// TIA Portal project "btvn_tuan2_light_traffic_2_chieu" (V14)

(* hardware
DEVICE "S7-1200 station_1"  S7-1200 Station
   slot 0: "Rack_0"  S7-1200 Rack  Rack  V1.0
   slot 1: "PLC_1"  CPU 1214C DC/DC/DC  6ES7 214-1AG40-0XB0  V4.2
DEVICE "HMI_1"  KTP700 Basic PN
   slot 0: "KTP700 Basic PN"  KTP700 Basic PN  6AV2 123-2GB03-0AX0  14.0.1.0
   slot 1: "HMI_RT_1"  KTP700 Basic PN  6AV2 123-2GB03-0AX0  14.0.1.0
   slot 5: "HMI_1.IE_CP_1"  PROFINET Interface  14.0.1.0
      slot 1: "PROFINET Interface_1"  PROFINET Interface
         slot 1: "Port_1"  Port
*)

// ===== PLC "PLC_1"  CPU 1214C DC/DC/DC =====

VAR_GLOBAL   // PLC tag table "Default tag table"
   "start" AT %M0.0 : Bool;
   "return" AT %M0.1 : Bool;
   "A do1" AT %M1.0 : Bool;
   "A vang1" AT %M1.2 : Bool;
   "A xanh 1" AT %M1.3 : Bool;
   "B do" AT %M0.5 : Bool;
   "B vang" AT %M0.6 : Bool;
   "B xanh" AT %M0.7 : Bool;
   "sleep mode" AT %I0.2 : Bool;
   "uu tien mode" AT %M1.1 : Bool;
   "uu tien 1" AT %I0.0 : Bool;
   "uu tien 2" AT %I0.1 : Bool;
   "tmp" AT %M1.4 : Bool;
   "tmp(1)" AT %M1.5 : Bool;
   "save2" AT %M1.6 : Bool;
   "save1" AT %M1.7 : Bool;
   "A vang 2" AT %M0.2 : Bool;
   "A xanh 2" AT %M0.3 : Bool;
   "A do 2" AT %M0.4 : Bool;
   "Tag_1" AT %Q0.2 : Bool;
   "Tag_2" AT %Q0.0 : Bool;
   "Tag_3" AT %Q0.1 : Bool;
   "Tag_4" AT %Q0.3 : Bool;
END_VAR

// folder: System blocks/Program resources

DATA_BLOCK "IEC_Timer_0_DB"   // DB1
{ S7_Optimized_Access := 'TRUE' }
AUTHOR : Simatic
FAMILY : IEC
NAME : IEC_TMR
VERSION : 1.0
// stored: InstanceOfName IEC_TIMER
"IEC_TIMER"
BEGIN
END_DATA_BLOCK

DATA_BLOCK "IEC_Timer_0_DB_1"   // DB2
{ S7_Optimized_Access := 'TRUE' }
AUTHOR : Simatic
FAMILY : IEC
NAME : IEC_TMR
VERSION : 1.0
// stored: InstanceOfName IEC_TIMER
"IEC_TIMER"
BEGIN
END_DATA_BLOCK

DATA_BLOCK "IEC_Timer_0_DB_2"   // DB3
{ S7_Optimized_Access := 'TRUE' }
AUTHOR : Simatic
FAMILY : IEC
NAME : IEC_TMR
VERSION : 1.0
// stored: InstanceOfName IEC_TIMER
"IEC_TIMER"
BEGIN
END_DATA_BLOCK

DATA_BLOCK "IEC_Timer_0_DB_3"   // DB4
{ S7_Optimized_Access := 'TRUE' }
AUTHOR : Simatic
FAMILY : IEC
NAME : IEC_TMR
VERSION : 1.0
// stored: InstanceOfName IEC_TIMER
"IEC_TIMER"
BEGIN
END_DATA_BLOCK

DATA_BLOCK "IEC_Timer_0_DB_4"   // DB5
{ S7_Optimized_Access := 'TRUE' }
AUTHOR : Simatic
FAMILY : IEC
NAME : IEC_TMR
VERSION : 1.0
// stored: InstanceOfName IEC_TIMER
"IEC_TIMER"
BEGIN
END_DATA_BLOCK

DATA_BLOCK "IEC_Timer_0_DB_5"   // DB6
{ S7_Optimized_Access := 'TRUE' }
AUTHOR : Simatic
FAMILY : IEC
NAME : IEC_TMR
VERSION : 1.0
// stored: InstanceOfName IEC_TIMER
"IEC_TIMER"
BEGIN
END_DATA_BLOCK

// folder: (top level)

ORGANIZATION_BLOCK "Main"   // OB1, LAD, ProgramCycle
TITLE = "Main Program Sweep (Cycle)"
{ S7_Optimized_Access := 'TRUE' }
VERSION : 0.1
   VAR_INPUT
      Initial_Call : Bool;   // Initial call of this OB
      Remanence : Bool;   // =True, if remanent data are available
   END_VAR
   VAR_TEMP   // added for the SCL form of the ladder/FBD networks
      _w1 : Bool;
   END_VAR
BEGIN

REGION Network 1: tuan tu sinh ra state den
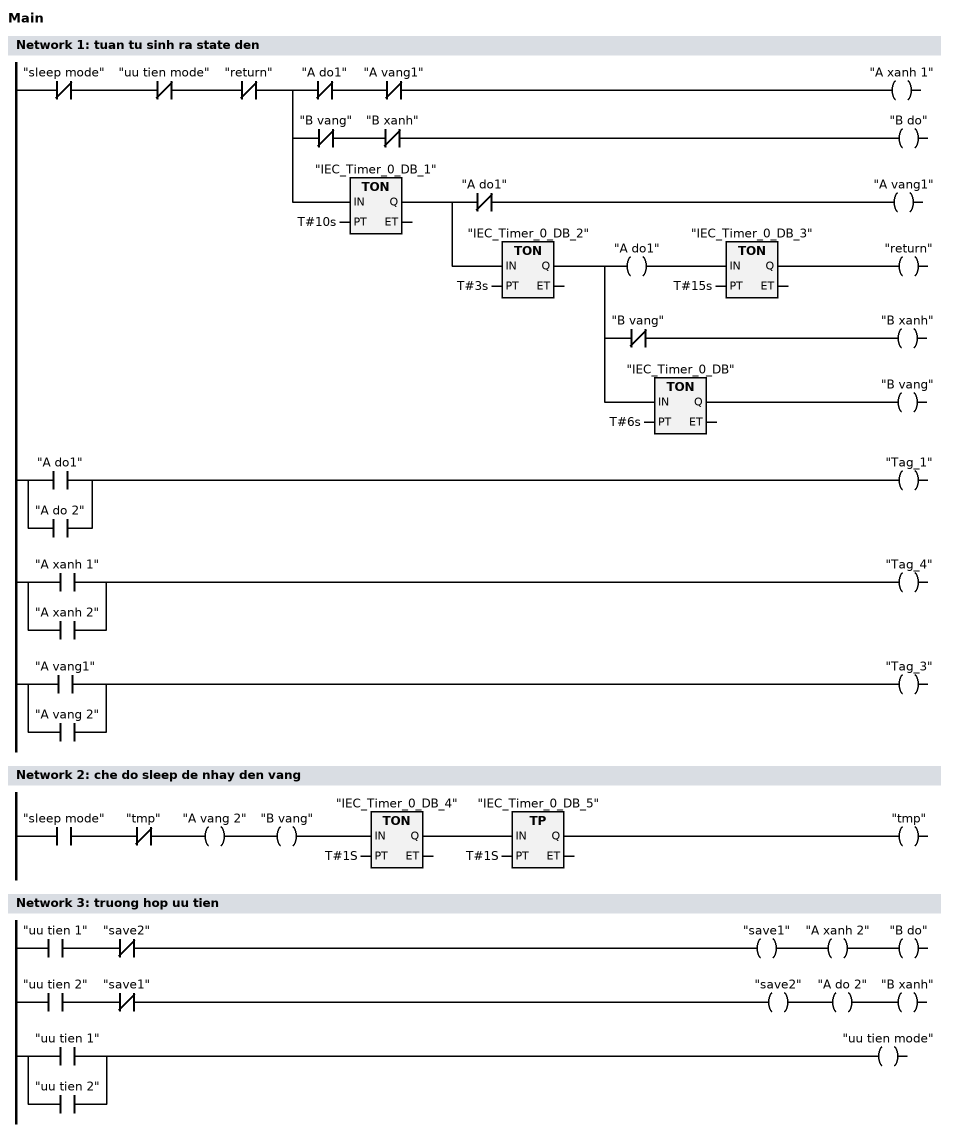
   #_w1 := NOT "sleep mode" AND NOT "uu tien mode" AND NOT "return";
   "A xanh 1" := #_w1 AND NOT "A do1" AND NOT "A vang1";
   "B do" := #_w1 AND NOT "B vang" AND NOT "B xanh";
   "IEC_Timer_0_DB_1".TON(IN := #_w1, PT := T#10s);
   "A vang1" := "IEC_Timer_0_DB_1".Q AND NOT "A do1";
   "IEC_Timer_0_DB_2".TON(IN := "IEC_Timer_0_DB_1".Q, PT := T#3s);
   "A do1" := "IEC_Timer_0_DB_2".Q;
   "IEC_Timer_0_DB_3".TON(IN := "IEC_Timer_0_DB_2".Q, PT := T#15s);
   "return" := "IEC_Timer_0_DB_3".Q;
   "B xanh" := "IEC_Timer_0_DB_2".Q AND NOT "B vang";
   "IEC_Timer_0_DB".TON(IN := "IEC_Timer_0_DB_2".Q, PT := T#6s);
   "B vang" := "IEC_Timer_0_DB".Q;
   "Tag_1" := "A do1" OR "A do 2";
   "Tag_4" := "A xanh 1" OR "A xanh 2";
   "Tag_3" := "A vang1" OR "A vang 2";
END_REGION

REGION Network 2: che do sleep de nhay den vang
   "A vang 2" := "sleep mode" AND NOT "tmp";
   "B vang" := "A vang 2";
   "IEC_Timer_0_DB_4".TON(IN := "A vang 2", PT := T#1S);
   "IEC_Timer_0_DB_5".TP(IN := "IEC_Timer_0_DB_4".Q, PT := T#1S);
   "tmp" := "IEC_Timer_0_DB_5".Q;
END_REGION

REGION Network 3: truong hop uu tien
   RUNG wire#powerrail
      Contact( "uu tien 1" )
      I_Contact( "save2" )
      Coil( "save1" )
      Coil( "A xanh 2" )
      Coil( "B do" )
   END_RUNG
   RUNG wire#powerrail
      Contact( "uu tien 2" )
      I_Contact( "save1" )
      Coil( "save2" )
      Coil( "A do 2" )
      Coil( "B xanh" )
   END_RUNG
   RUNG wire#powerrail
      Contact( "uu tien 1" )
      wire#w1
      Coil( "uu tien mode" )
   END_RUNG
   RUNG wire#powerrail
      Contact( "uu tien 2" )
   END_RUNG wire#w1
   // the same network as SCL:
   "save1" := "uu tien 1" AND NOT "save2";
   "A xanh 2" := "save1";
   "B do" := "save1";
   "save2" := "uu tien 2" AND NOT "save1";
   "A do 2" := "save2";
   "B xanh" := "save2";
   "uu tien mode" := "uu tien 1" OR "uu tien 2";
END_REGION
END_ORGANIZATION_BLOCK

(* ===== HMI "HMI_RT_1" =====
system functions are stored by id; their names below are inferred from use
connection "HMI_Connection_1": ETHERNET, SMART_S7_1200_OMS

HMI tags "Default tag table"
   "Tag_ScreenNumber" : UInt, internal
   "sleep mode" : Bool = PLC "sleep mode" AT %I0.2, 1 s
   "uu tien 1" : Bool = PLC "uu tien 1" AT %I0.0, 1 s
   "uu tien 2" : Bool = PLC "uu tien 2" AT %I0.1, 1 s
   "A xanh 1" : Bool = PLC "A xanh 1" AT %M1.3, 1 s
   "A vang1" : Bool = PLC "A vang1" AT %M1.2, 1 s
   "A do1" : Bool = PLC "A do1" AT %M1.0, 1 s
   "B xanh" : Bool = PLC "B xanh" AT %M0.7, 1 s
   "B vang" : Bool = PLC "B vang" AT %M0.6, 1 s
   "B do" : Bool = PLC "B do" AT %M0.5, 1 s

Template "Template_1" 800x480
   Button "Exit" at 714,429 size 71x50; TextOff 'Exit'; PictureOff "ExitRuntime_KTP700_Basic_PN_TR"; PictureOn "ExitRuntime_KTP700_Basic_PN_TR"
      on Release: StopRuntime(0)
   Button "Template_Button" at 614,429 size 71x50; TextOff 'Text'
   Button "Template_Button_1" at 514,429 size 71x50; TextOff 'Text'
   Button "Template_Button_2" at 414,429 size 71x50; TextOff 'Text'
   Button "Template_Button_3" at 314,429 size 71x50; TextOff 'Text'
   Button "Template_Button_4" at 214,429 size 71x50; TextOff 'Text'
   Button "Alarms" at 114,429 size 71x50; TextOff 'Alarms'; PictureOff "AlarmDisplay_KTP700_Basic_PN_TR"; PictureOn "AlarmDisplay_KTP700_Basic_PN_TR"
      on Release: function_ef3f5d25("Alarm window_Unacknowledged", -1)
   Button "Start screen" at 14,429 size 71x50; TextOff 'Start screen'; PictureOff "NavigateHome_KTP700_Basic_PN_TR"; PictureOn "NavigateHome_KTP700_Basic_PN_TR"
      on Release: ActivateScreen("Root screen", 0)
   SymbolicIOField "Symbolic_IO_Field_Screen" at 93,9 size 600x33; TextOff '0'; TextOn '1'; TextList "TextList_ScreenNames"
      ProcessValue <- "Tag_ScreenNumber"
      on Change: ActivateScreenByNumber("Tag_ScreenNumber", 0)
   DateTimeField "HmiScreenItemData" at 695,25 size 105x25
   DateTimeField "HmiScreenItemData_1" at 695,0 size 105x25
   GraphicView "Logo" at 0,0 size 91x51; Picture "Logo of HMI_1"

screen "Root screen" 800x480, template "Template_1"
   on GenerateScreen: SetTag("Tag_ScreenNumber", 1)
   Circle "Circle_1" at 381,18 size 23x23
      Appearance <- "A xanh 1"
   Circle "Circle_2" at 381,45 size 23x23
      Appearance <- "A vang1"
   Circle "Circle_3" at 381,75 size 23x23
      Appearance <- "A do1"
   Circle "Circle_4" at 398,233 size 23x23
      Appearance <- "B xanh"
   Circle "Circle_5" at 398,260 size 23x23
      Appearance <- "B vang"
   Circle "Circle_6" at 398,290 size 23x23
      Appearance <- "B do"
   Switch "Switch_1" at 4,123 size 64x32; TextOn 'ON'; CaptionText 'Switch'; TextOff 'OFF'
      on SwitchOff: ResetBit("sleep mode")
      on SwitchOn: SetBit("sleep mode")
   TextField "Text field_1" at 83,118 size 46x23; Text 'Daily'
   TextField "Text field_2" at 83,138 size 51x23; Text 'warm'
   Switch "Switch_3" at 265,33 size 64x32; TextOn 'ON'; CaptionText 'Switch'; TextOff 'OFF'
      on SwitchOn: SetBit("uu tien 1")
      on SwitchOff: ResetBit("uu tien 1")
   Switch "Switch_4" at 293,364 size 64x32; TextOn 'ON'; CaptionText 'Switch'; TextOff 'OFF'
      on SwitchOn: SetBit("uu tien 2")
      on SwitchOff: ResetBit("uu tien 2")
*)